// Mitsubishi GX Developer project: 16-505   PLC: FX1S

PROGRAM MAIN
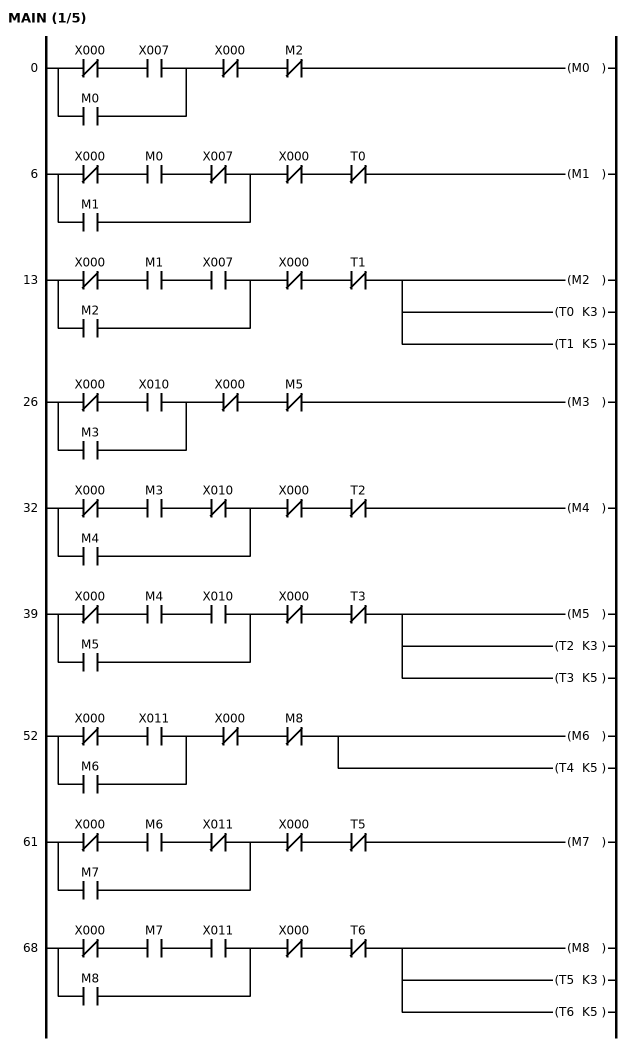
0     LDI     X000
      AND     X007
      OR      M0
      ANI     X000
      ANI     M2
      OUT     M0
6     LDI     X000
      AND     M0
      ANI     X007
      OR      M1
      ANI     X000
      ANI     T0
      OUT     M1
13    LDI     X000
      AND     M1
      AND     X007
      OR      M2
      ANI     X000
      ANI     T1
      OUT     M2
      OUT     T0 K3
      OUT     T1 K5
26    LDI     X000
      AND     X010
      OR      M3
      ANI     X000
      ANI     M5
      OUT     M3
32    LDI     X000
      AND     M3
      ANI     X010
      OR      M4
      ANI     X000
      ANI     T2
      OUT     M4
39    LDI     X000
      AND     M4
      AND     X010
      OR      M5
      ANI     X000
      ANI     T3
      OUT     M5
      OUT     T2 K3
      OUT     T3 K5
52    LDI     X000
      AND     X011
      OR      M6
      ANI     X000
      ANI     M8
      OUT     M6
      OUT     T4 K5
61    LDI     X000
      AND     M6
      ANI     X011
      OR      M7
      ANI     X000
      ANI     T5
      OUT     M7
68    LDI     X000
      AND     M7
      AND     X011
      OR      M8
      ANI     X000
      ANI     T6
      OUT     M8
      OUT     T5 K3
      OUT     T6 K5
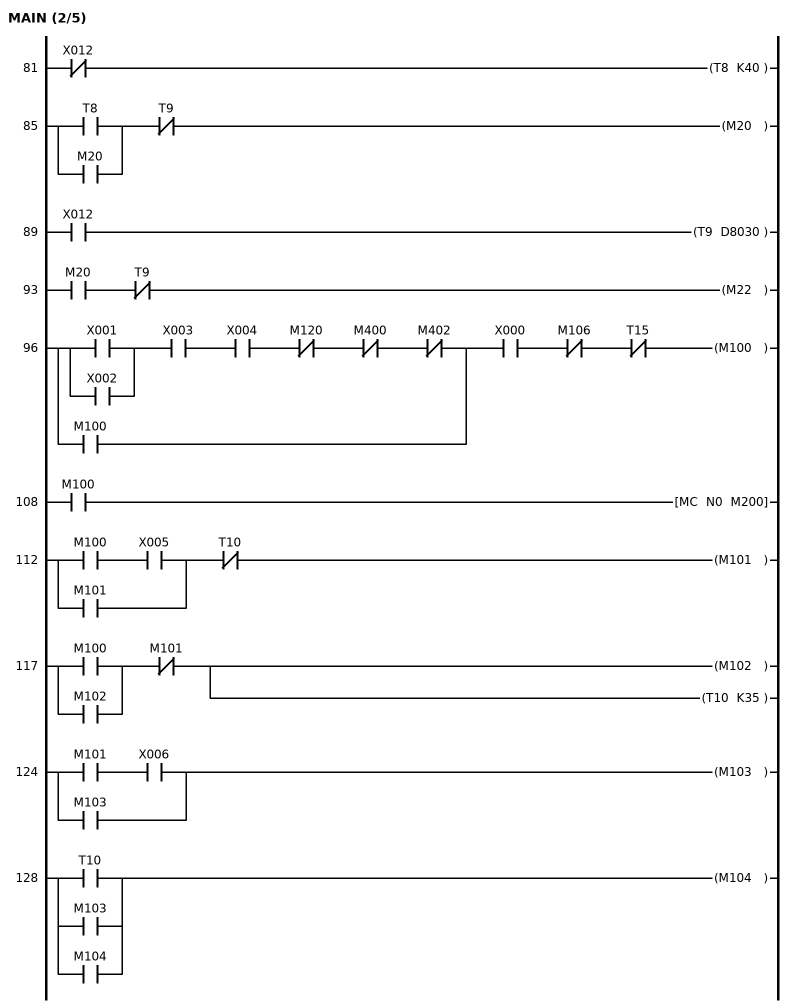
81    LDI     X012
      OUT     T8 K40
85    LD      T8
      OR      M20
      ANI     T9
      OUT     M20
89    LD      X012
      OUT     T9 D8030
93    LD      M20
      ANI     T9
      OUT     M22
96    LD      X001
      OR      X002
      AND     X003
      AND     X004
      ANI     M120
      ANI     M400
      ANI     M402
      OR      M100
      AND     X000
      ANI     M106
      ANI     T15
      OUT     M100
108   LD      M100
      MC      N0 M200
112   LD      M100
      AND     X005
      OR      M101
      ANI     T10
      OUT     M101
117   LD      M100
      OR      M102
      ANI     M101
      OUT     M102
      OUT     T10 K35
124   LD      M101
      AND     X006
      OR      M103
      OUT     M103
128   LD      T10
      OR      M103
      OR      M104
      OUT     M104
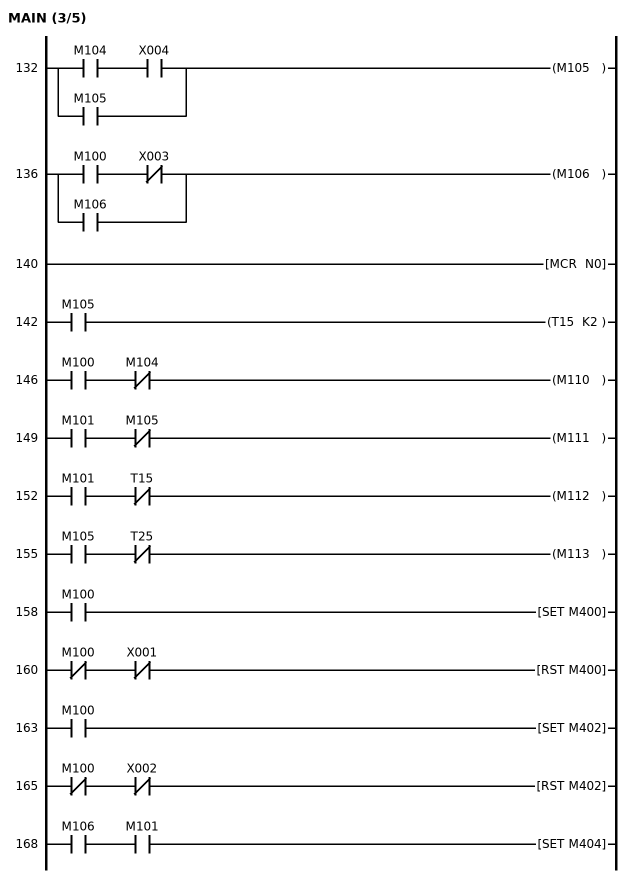
132   LD      M104
      AND     X004
      OR      M105
      OUT     M105
136   LD      M100
      ANI     X003
      OR      M106
      OUT     M106
140   MCR     N0
142   LD      M105
      OUT     T15 K2
146   LD      M100
      ANI     M104
      OUT     M110
149   LD      M101
      ANI     M105
      OUT     M111
152   LD      M101
      ANI     T15
      OUT     M112
155   LD      M105
      ANI     T25
      OUT     M113
158   LD      M100
      SET     M400
160   LDI     M100
      ANI     X001
      RST     M400
163   LD      M100
      SET     M402
165   LDI     M100
      ANI     X002
      RST     M402
168   LD      M106
      AND     M101
      SET     M404
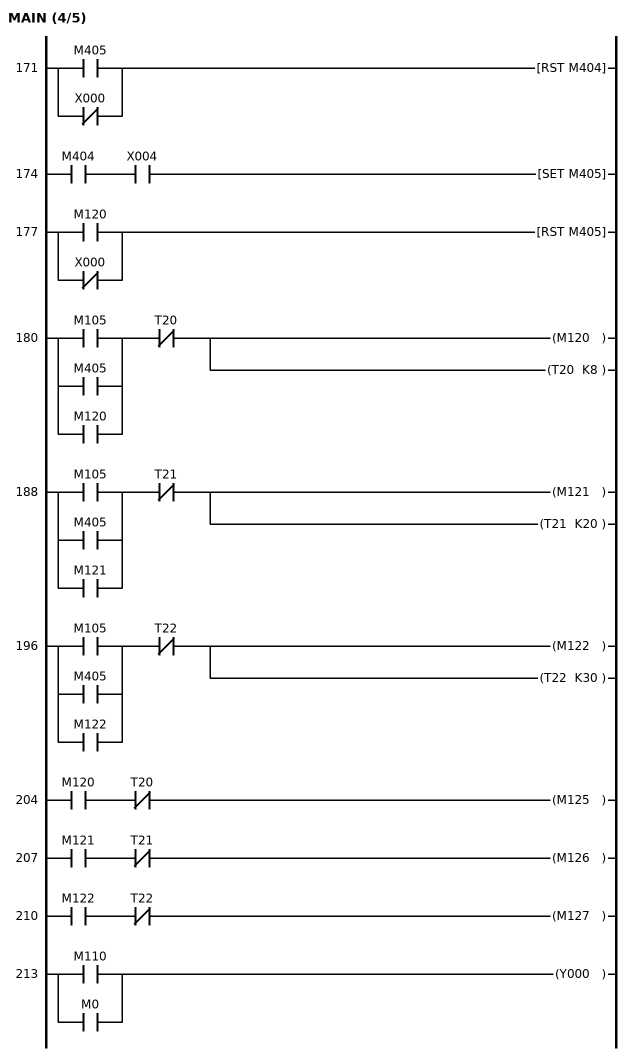
171   LD      M405
      ORI     X000
      RST     M404
174   LD      M404
      AND     X004
      SET     M405
177   LD      M120
      ORI     X000
      RST     M405
180   LD      M105
      OR      M405
      OR      M120
      ANI     T20
      OUT     M120
      OUT     T20 K8
188   LD      M105
      OR      M405
      OR      M121
      ANI     T21
      OUT     M121
      OUT     T21 K20
196   LD      M105
      OR      M405
      OR      M122
      ANI     T22
      OUT     M122
      OUT     T22 K30
204   LD      M120
      ANI     T20
      OUT     M125
207   LD      M121
      ANI     T21
      OUT     M126
210   LD      M122
      ANI     T22
      OUT     M127
213   LD      M110
      OR      M0
      OUT     Y000
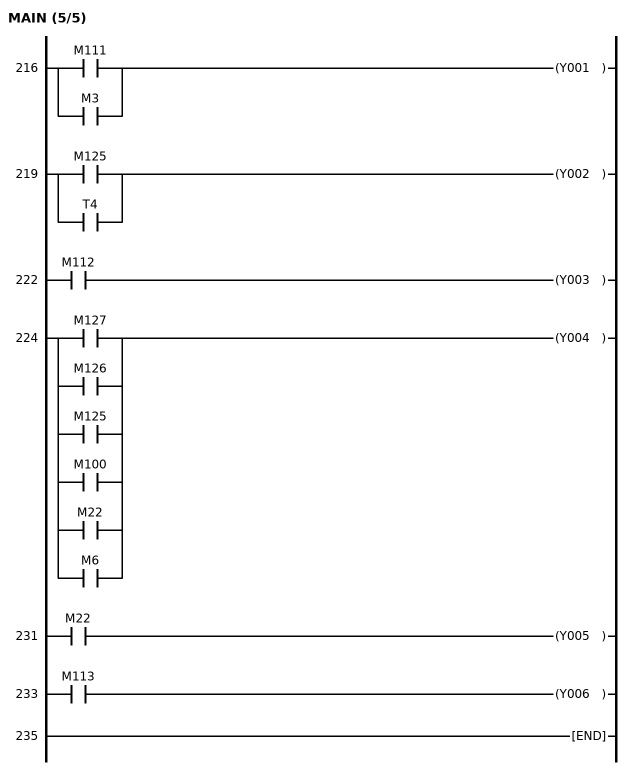
216   LD      M111
      OR      M3
      OUT     Y001
219   LD      M125
      OR      T4
      OUT     Y002
222   LD      M112
      OUT     Y003
224   LD      M127
      OR      M126
      OR      M125
      OR      M100
      OR      M22
      OR      M6
      OUT     Y004
231   LD      M22
      OUT     Y005
233   LD      M113
      OUT     Y006
235   END
END_PROGRAM
